// LS Electric XG5000 project: 유튜브방송용_2021082820
// PLC NewPLC

PROGRAM NewProgram (task: 스캔 프로그램)

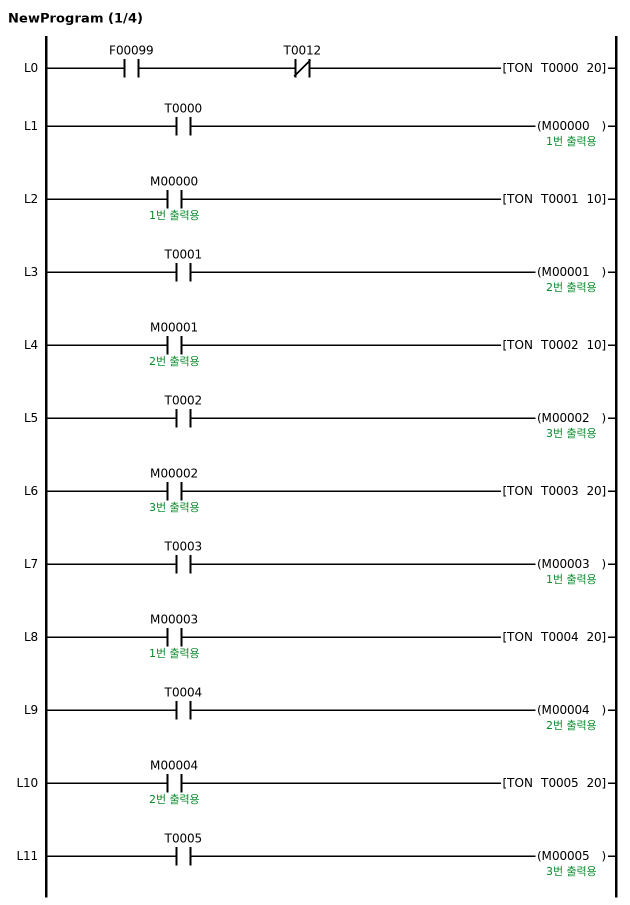
; L0
LOAD      F00099
AND NOT   T0012
TON       T0000 20
; L1
LOAD      T0000
OUT       M00000	// 1번 출력용
; L2
LOAD      M00000	// 1번 출력용
TON       T0001 10
; L3
LOAD      T0001
OUT       M00001	// 2번 출력용
; L4
LOAD      M00001	// 2번 출력용
TON       T0002 10
; L5
LOAD      T0002
OUT       M00002	// 3번 출력용
; L6
LOAD      M00002	// 3번 출력용
TON       T0003 20
; L7
LOAD      T0003
OUT       M00003	// 1번 출력용
; L8
LOAD      M00003	// 1번 출력용
TON       T0004 20
; L9
LOAD      T0004
OUT       M00004	// 2번 출력용
; L10
LOAD      M00004	// 2번 출력용
TON       T0005 20
; L11
LOAD      T0005
OUT       M00005	// 3번 출력용

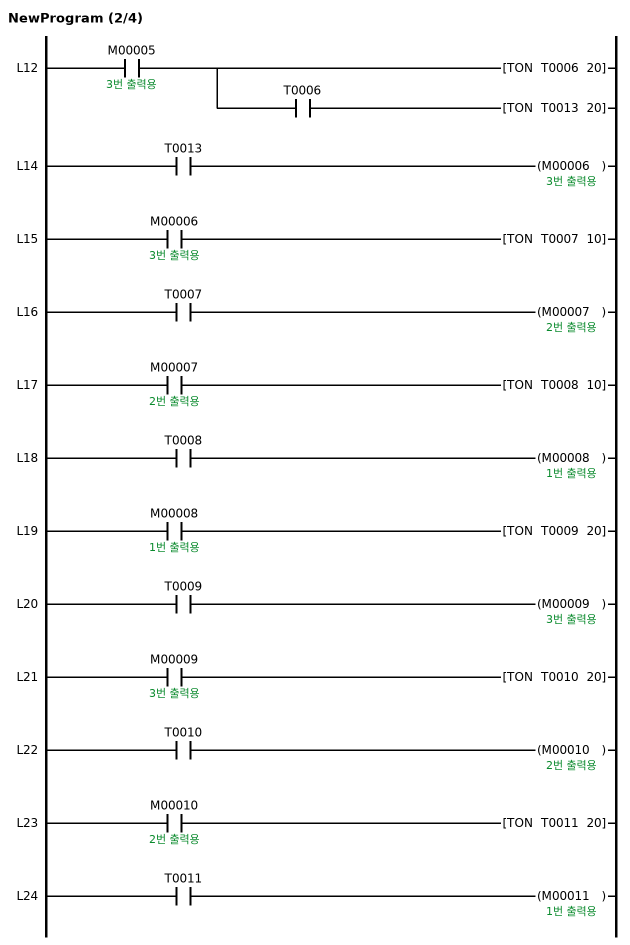
; L12
LOAD      M00005	// 3번 출력용
TON       T0006 20
AND       T0006
TON       T0013 20
; L14
LOAD      T0013
OUT       M00006	// 3번 출력용
; L15
LOAD      M00006	// 3번 출력용
TON       T0007 10
; L16
LOAD      T0007
OUT       M00007	// 2번 출력용
; L17
LOAD      M00007	// 2번 출력용
TON       T0008 10
; L18
LOAD      T0008
OUT       M00008	// 1번 출력용
; L19
LOAD      M00008	// 1번 출력용
TON       T0009 20
; L20
LOAD      T0009
OUT       M00009	// 3번 출력용
; L21
LOAD      M00009	// 3번 출력용
TON       T0010 20
; L22
LOAD      T0010
OUT       M00010	// 2번 출력용
; L23
LOAD      M00010	// 2번 출력용
TON       T0011 20
; L24
LOAD      T0011
OUT       M00011	// 1번 출력용

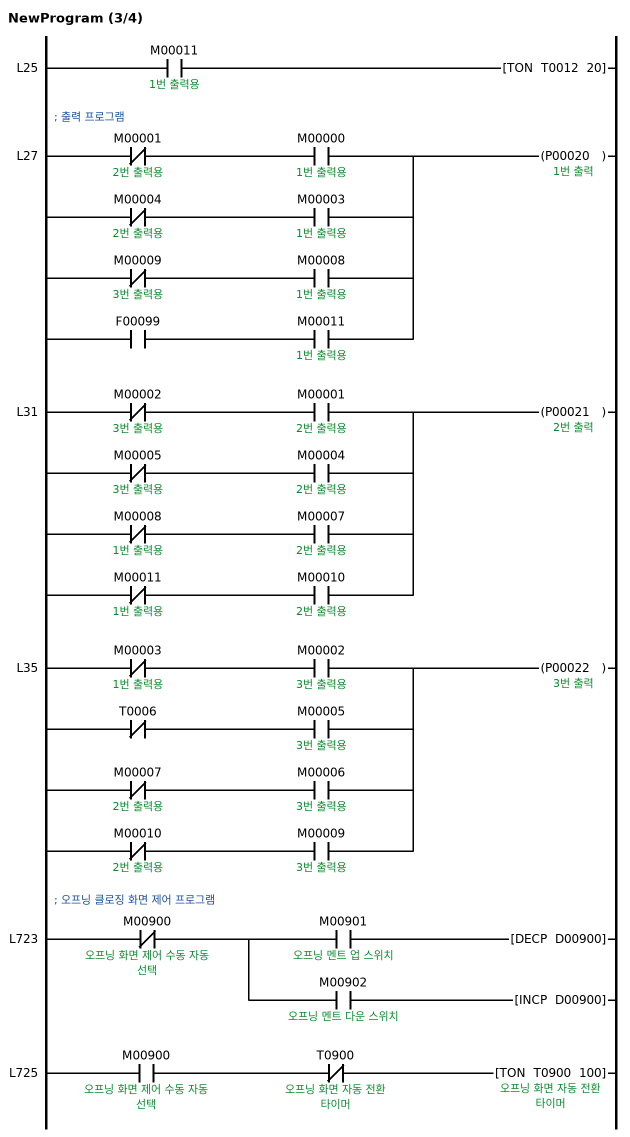
; L25
LOAD      M00011	// 1번 출력용
TON       T0012 20
// 출력 프로그램
; L27
LOAD NOT  M00001	// 2번 출력용
AND       M00000	// 1번 출력용
LOAD NOT  M00004	// 2번 출력용
AND       M00003	// 1번 출력용
OR LOAD
LOAD NOT  M00009	// 3번 출력용
AND       M00008	// 1번 출력용
OR LOAD
LOAD      F00099
AND       M00011	// 1번 출력용
OR LOAD
OUT       P00020	// 1번 출력
; L31
LOAD NOT  M00002	// 3번 출력용
AND       M00001	// 2번 출력용
LOAD NOT  M00005	// 3번 출력용
AND       M00004	// 2번 출력용
OR LOAD
LOAD NOT  M00008	// 1번 출력용
AND       M00007	// 2번 출력용
OR LOAD
LOAD NOT  M00011	// 1번 출력용
AND       M00010	// 2번 출력용
OR LOAD
OUT       P00021	// 2번 출력
; L35
LOAD NOT  M00003	// 1번 출력용
AND       M00002	// 3번 출력용
LOAD NOT  T0006
AND       M00005	// 3번 출력용
OR LOAD
LOAD NOT  M00007	// 2번 출력용
AND       M00006	// 3번 출력용
OR LOAD
LOAD NOT  M00010	// 2번 출력용
AND       M00009	// 3번 출력용
OR LOAD
OUT       P00022	// 3번 출력
// 오프닝 클로징 화면 제어 프로그램
; L723
LOAD NOT  M00900	// 오프닝 화면 제어 수동 자동 선택
MPUSH
AND       M00901	// 오프닝 멘트 업 스위치
DECP      D00900
MPOP
AND       M00902	// 오프닝 멘트 다운 스위치
INCP      D00900
; L725
LOAD      M00900	// 오프닝 화면 제어 수동 자동 선택
AND NOT   T0900	// 오프닝 화면 자동 전환 타이머
TON       T0900 100	// 오프닝 화면 자동 전환 타이머

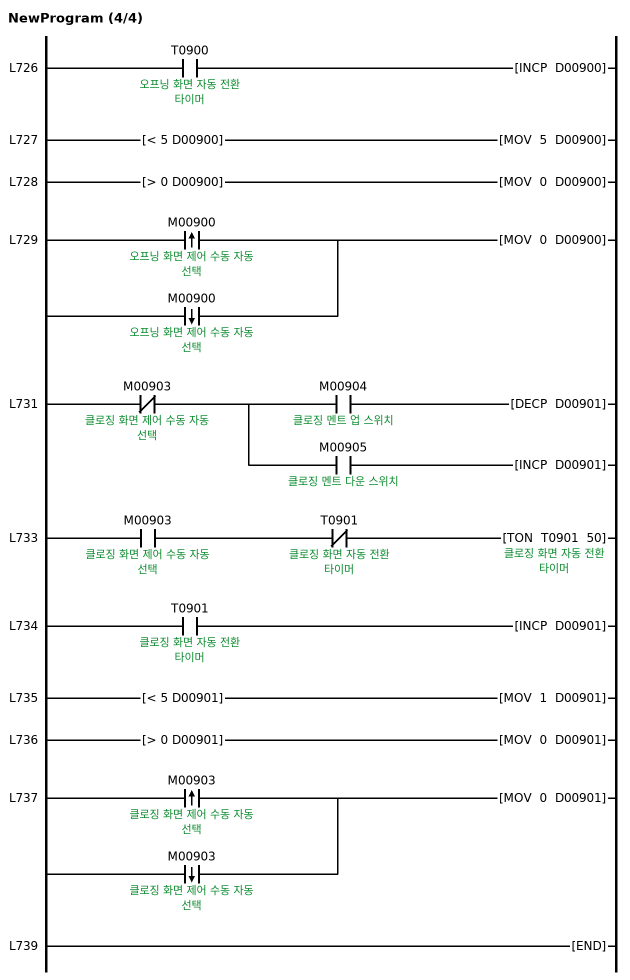
; L726
LOAD      T0900	// 오프닝 화면 자동 전환 타이머
INCP      D00900
; L727
LOAD<     5 D00900
MOV       5 D00900
; L728
LOAD>     0 D00900
MOV       0 D00900
; L729
LOADP     M00900	// 오프닝 화면 제어 수동 자동 선택
ORN       M00900	// 오프닝 화면 제어 수동 자동 선택
MOV       0 D00900
; L731
LOAD NOT  M00903	// 클로징 화면 제어 수동 자동 선택
MPUSH
AND       M00904	// 클로징 멘트 업 스위치
DECP      D00901
MPOP
AND       M00905	// 클로징 멘트 다운 스위치
INCP      D00901
; L733
LOAD      M00903	// 클로징 화면 제어 수동 자동 선택
AND NOT   T0901	// 클로징 화면 자동 전환 타이머
TON       T0901 50	// 클로징 화면 자동 전환 타이머
; L734
LOAD      T0901	// 클로징 화면 자동 전환 타이머
INCP      D00901
; L735
LOAD<     5 D00901
MOV       1 D00901
; L736
LOAD>     0 D00901
MOV       0 D00901
; L737
LOADP     M00903	// 클로징 화면 제어 수동 자동 선택
ORN       M00903	// 클로징 화면 제어 수동 자동 선택
MOV       0 D00901
; L739
END